Omron Sysmac Studio project ISA_T4Q5_a (Sysmac Studio 1.23.0.14, StandardProject)

# Controller new_Controller_0: NX1P2-1040DT1 version 1.18
Task PrimaryTask (priority 4, period or condition 8000): Programa0
Library INV00x_MX2_ECT 1.0.9 (contents left out)

VAR_GLOBAL
    PP : BOOL;  (* at BuiltInIO://cpu/#0/Input_Bit_00 *)
    PM : BOOL;  (* at BuiltInIO://cpu/#0/Input_Bit_01 *)
    Variador_01_Comando : WORD;  (* at ECAT://node#11/Command *)
    Variador_01_Frecuencia : UINT;  (* at ECAT://node#11/Frequency reference *)
    presion_raw : INT;  (* at BuiltInIO://opt/#0/Ch1_Analog_Input_Value *)
    PP_VAR : BOOL;
    PM_VAR : BOOL;
    PP_HMI AT %W0.00 : BOOL;  (* published *)
    PM_HMI AT %W0.01 : BOOL;  (* published *)
END_VAR
VAR_GLOBAL RETAIN
    presion_real AT %D0 : REAL;  (* published *)
    caudal_real AT %D2 : REAL;  (* published *)
END_VAR

PROGRAM Programa0
VAR
    presion_limitada : REAL;
END_VAR
VAR CONSTANT
    caudal_a_50Hz : REAL := 0.5;
END_VAR
VAR
    frecuencia_real : REAL;
    presion_raw_limitada : INT;
END_VAR
VAR_EXTERNAL
    PM : BOOL;
    Variador_01_Comando : WORD;
    PP : BOOL;
    Variador_01_Frecuencia : UINT;
    presion_raw : INT;
    PP_VAR : BOOL;
    PM_VAR : BOOL;
    PM_HMI : BOOL;
    presion_real : REAL;
    caudal_real : REAL;
    PP_HMI : BOOL;
END_VAR

(* Section calculos: ladder, written here as Structured Text *)

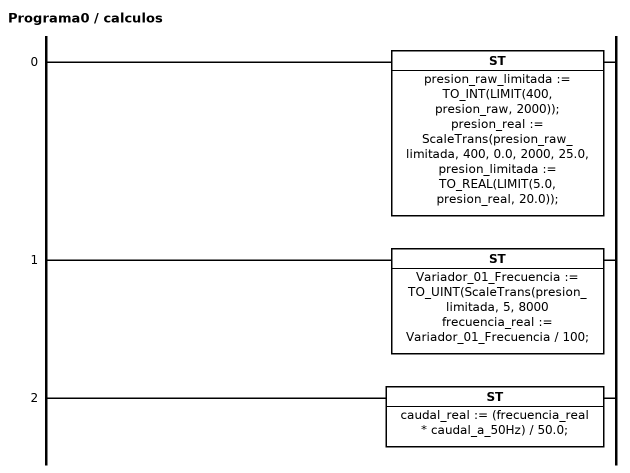
(* Rung 0 *)
presion_raw_limitada := TO_INT(LIMIT(400, presion_raw, 2000));
presion_real := ScaleTrans(presion_raw_limitada, 400, 0.0, 2000, 25.0, 0.0);
presion_limitada := TO_REAL(LIMIT(5.0, presion_real, 20.0));
(* Rung 1 *)
Variador_01_Frecuencia := TO_UINT(ScaleTrans(presion_limitada, 5, 8000, 20, 0, 0));
frecuencia_real := Variador_01_Frecuencia / 100;
(* Rung 2 *)
caudal_real := (frecuencia_real * caudal_a_50Hz) / 50.0;

(* Section principal: ladder, written here as Structured Text *)

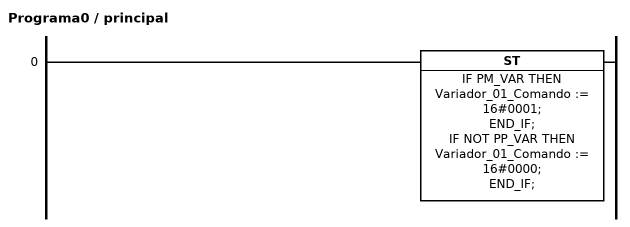
(* Rung 0 *)
IF PM_VAR THEN
	Variador_01_Comando := 16#0001;
END_IF;

IF NOT PP_VAR THEN
	Variador_01_Comando := 16#0000;
END_IF;

(* Section hmi_plc: ladder, written here as Structured Text *)

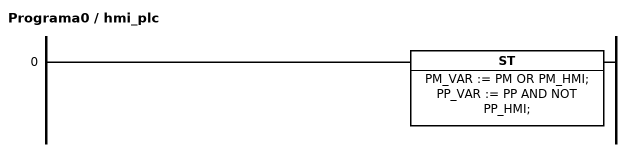
(* Rung 0 *)
PM_VAR := PM OR PM_HMI;
PP_VAR := PP AND NOT PP_HMI;
END_PROGRAM